FUNCTION_BLOCK LOAD_CTL (* Workpiece LOAD Solenoid Control *)
  (* Standard: 61499-1; Classification: Simulation; ApplicationDomain: Material Handling; Function: Control; Type: Workpiece Loading *)
  (* Version 0.2, 2002-07-16, JHC, Rockwell Automation, Changed back to LD with IND triggering in ECC. *)
  (* Version 0.1, 2002-05-24, JHC, Rockwell Automation, Changed from LD to FBD to get E_D_FF triggering. *)
  (* Version 0.0, 2002-05-20, JHC, Rockwell Automation, Copied/Modified from XBAR_CTL. *)
  (* Compiler header: package fb.rt.mach; import fb.rt.math.*; *)
  (* Compiler Java IBM Jikes 1.06 *)
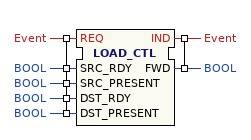
  EVENT_INPUT
    REQ WITH SRC_RDY, SRC_PRESENT, DST_RDY, DST_PRESENT;
  END_EVENT
  EVENT_OUTPUT
    IND WITH FWD; (* Change in FWD output *)
  END_EVENT
  VAR_INPUT
    SRC_RDY : BOOL; (* Source in position for transfer *)
    SRC_PRESENT : BOOL; (* Workpiece present at source *)
    DST_RDY : BOOL; (* Destination in position for transfer *)
    DST_PRESENT : BOOL; (* Workpiece present at destination *)
  END_VAR
  VAR_OUTPUT
    FWD : BOOL; (* Actuator direction:1=FWD,0=REV *)
  END_VAR
  VAR
    WAS_FWD : BOOL;
  END_VAR
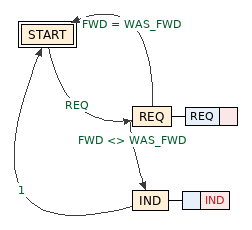
  EC_STATES
    START;
    REQ : REQ;
    IND : -> IND;
  END_STATES
  EC_TRANSITIONS
    START TO REQ := REQ;
    REQ TO START := FWD = WAS_FWD;
    REQ TO IND := FWD <> WAS_FWD;
    IND TO START := 1;
  END_TRANSITIONS
  ALGORITHM REQ IN LD:
    WAS_FWD := FWD;
    FWD := SRC_RDY SRC_PRESENT & DST_RDY & DST_PRESENT ! &;
  END_ALGORITHM
END_FUNCTION_BLOCK
